Staubli VAL3: FC_EndMotion.pgx

program FC_EndMotion()
begin
  //this function is to finish the synchronous motion
  $movejSyncEnd()
  //delay(5)
  //sScrPts="NOT READY"
  //n_sTxt=0
end
